{attribute 'pack_mode' := '1'}
    {attribute 'OPC.UA.DA' := '1'}
    {attribute 'OPC.UA.DA.StructuredType' := '1'}
    (*
    ST_RW_Digital_In_HMI_IgnitionExp
    ==================================================
    Generated from Ignition UDT: RW_Digital_In
    Total tags: 5
    Generated on: 2025-09-16 15:04:58
    *)
    TYPE ST_RW_Digital_In_HMI_IgnitionExp :
    STRUCT
        {attribute 'OPC.UA.DA' := '1'}
        Manual_Input : BOOL := FALSE;
        {attribute 'OPC.UA.DA' := '1'}
        AllowManualOverride : BOOL := FALSE;
        {attribute 'OPC.UA.DA' := '1'}
        Manual_Mode : BOOL := FALSE;
        {attribute 'OPC.UA.DA' := '1'}
        Input_Raw : BOOL := FALSE;
        {attribute 'OPC.UA.DA' := '1'}
        Input : BOOL := FALSE;
    END_STRUCT
    END_TYPE

(* stored: Version 1.1.0.1
   DUT ST_RW_Digital_In_HMI_IgnitionExp: Id {6411c3ac-6e7b-425f-8089-9a175b22060b} *)
